FUNCTION_BLOCK PUBLIC ABSTRACT TcoTaskedSequencer EXTENDS TcoCore.TcoSequencerBase
VAR
	{attribute addProperty Name "|[[1]AttributeName]|"}
	{attribute addProperty ToolTip "|[[1]AttributeToolTip]|"}
    _task : TcoInnerTask(THIS^);
    _o    : TcoCore.TcoSequencerObserver(THIS^);	
	
	{attribute addProperty Name "|[[1]Cycle Time Analitics]|"} 
	_cycleTimeAnalitics:CycleTimeAnalitics;	
	_startCleanCycleTime: TIME;
	_stopCleanCycleTime: TIME;
	_timer_1: TON;
	_timer_2: TON;
	_detectStartSeq : R_TRIG;

	_customObserver:TcoCustomSequencerObserver(THIS^);
END_VAR

Run();

PROPERTY PUBLIC AverageCleanCycleTime : TIME
GET
AverageCleanCycleTime:=_cycleTimeAnalitics.AverageCleanCycle;
END_GET
END_PROPERTY

PROPERTY PUBLIC AverageCycleTime : TIME
GET
AverageCycleTime:=_cycleTimeAnalitics.Average;
END_GET
END_PROPERTY

(*~
	<docu>
		<summary>
			Completes the actually running step, when the `inCondition` parameter is `TRUE`.
			Method is typically called inside a step as the transition method.
		</summary>			
	</docu>	
~*)
METHOD PROTECTED FINAL Await
VAR_INPUT
    (*~
	<docu>
		<summary>
			The condition under which the step is completed.
		</summary>			
	</docu>	
~*)
    inCondition : BOOL;
END_VAR
i_StepCompleteWhen(inCondition := inCondition);
END_METHOD

(*~
	<docu>
		<summary>
			<para>
				Completes the sequencer, and return the sequencer pointer to the first step in the seuqence.
				Method is typically called inside the last step of the sequence.
			</para>
		</summary>			
	</docu>	
~*)
METHOD PROTECTED FINAL CompleteSequence



i_CompleteSequence();

IF _cycleTimeAnalitics.FilterConstant = 0 THEN;
	_cycleTimeAnalitics.FilterConstant:=10;
END_IF;


IF _cycleTimeAnalitics.Average = T#0S THEN
	_cycleTimeAnalitics.Average:=_SequenceElapsedTime;
END_IF
_cycleTimeAnalitics.Average:= (((_cycleTimeAnalitics.FilterConstant-1)*_cycleTimeAnalitics.Average)+_LastCycleTime)/_cycleTimeAnalitics.FilterConstant;

_startCleanCycleTime:=T#0S;
_stopCleanCycleTime:=T#0S;
END_METHOD

(*~
	<docu>
		<summary>
			Completes the execution of the current step and moves the sequencer pointer to the next step in order of execution.
			The call returns `ITcoObjectRestorer` that allows to restore object upon step completition.
		</summary>		
		<returns></returns>	
	</docu>	
~*)
METHOD PROTECTED FINAL CompleteStep : ITcoObjectRestorer

CompleteStep := i_CompleteStep();
END_METHOD

PROPERTY CustomObserver : REFERENCE TO TcoCustomSequencerObserver
GET
CustomObserver ref= _customObserver;
END_GET
END_PROPERTY

PROPERTY PUBLIC CycleTimeFilterConstant : UINT
GET
CycleTimeFilterConstant:=_cycleTimeAnalitics.FilterConstant;
END_GET
SET // PUBLIC
_cycleTimeAnalitics.FilterConstant:=CycleTimeFilterConstant;
END_SET
END_PROPERTY

(*~
	<docu>
		<summary>
			Main method of the sequener. Custom code needs to be placed here. The sequencer is executed by call of **Instance.Run()** method.
			This method is abstract, and it must be overridden in derived block.
		</summary>
	</docu>
~*)
METHOD PROTECTED  Main : BOOL
END_METHOD

(*~
	<docu>
		<summary>
			Completes the execution of the current step and moves the sequencer pointer to the next step in order of execution.
			The call returns `ITcoObjectRestorer` that allows to restore object upon step completition.
		</summary>		
		<returns></returns>	
	</docu>	
~*)
METHOD PROTECTED FINAL Next : ITcoObjectRestorer
Next := i_CompleteStep();
END_METHOD

METHOD PUBLIC OnAbort : BOOL
SUPER^.Restore();
END_METHOD

METHOD PUBLIC OnDone : BOOL
END_METHOD

METHOD PUBLIC OnError : BOOL
END_METHOD


(*~
	<docu>
		<summary>
			This method is called on sequence completion (the sequencer's last step was completed). 
			This method can be overridden in derived block with a custom logic.
		</summary>			
	</docu>	
~*)
METHOD PROTECTED OnSequenceCompleted
SUPER^.OnSequenceCompleted();
_customObserver.DefineEndTime(Context.RealTimeClock.NowLocalAsTIMESTRUCT());
_customObserver.CompleteSequence();
END_METHOD

METHOD PUBLIC OnStart
_startCleanCycleTime:=T#0S;
_stopCleanCycleTime:=T#0S;
END_METHOD

(*~
	<docu>
		<summary>
			This method is executed upon step completion.
			This method can be overridden in derived block by custom logic.
		</summary>			
	</docu>	
~*)
METHOD PROTECTED OnStepCompleted


_customObserver.Observe(
	inID:= _currentStep.ID, 
	inDescription:= _currentStep.Description, 
	inDuration:= _currentStep.Duration);
END_METHOD

METHOD pr_Close
VAR_INPUT
END_VAR
_lastClosingCycle := Context.StartCycleCount;

IF _sequencerHasError THEN
    OnSequencerError(_sequencerErrorId);
END_IF

_previousNumberOfStepsInSequence := _numberOfStepsInSequence;
Context.Environment.Messaging.Suspend();

IF _modeController._stepIn.Done THEN
    _modeController._stepIn.Restore();
END_IF

Context.Environment.Messaging.Resume();

_restoringSequence := FALSE;
END_METHOD

METHOD pr_Open
VAR
    _message : STRING(255);
END_VAR
_theOrderOfTheCurrentlyEvaluatedStep := 0;

IF _requestStepActive AND
    _requestedStepId <> (MinStepID - 1) AND
    (_modeController.Mode <> eSequencerMode.StepMode OR _modeController._stepIn.Busy OR _checkStepIdRequestedInStepMode) THEN
    _requestStepCycle := _requestStepCycle + 1;
ELSE
    _requestStepCycle := 0;

END_IF

IF _requestStepCycle > 1 AND NOT _sequencerHasError THEN
    _sequencerErrorId        := eSequencerError.StepWithRequestedIdDoesNotExists;
    _message                 := CONCAT('REQUESTED STEP_ID: ', INT_TO_STRING(_requestedStepId));
    _message                 := CONCAT(_message, ' DOES NOT EXIST');
    _currentStep.Description := _message;
    _currentStep.Status      := eStepStatus.Error;
    THIS^.Messenger.Post(_message, eMessageCategory.ProgrammingError);
    _sequencerHasError := TRUE;

END_IF

IF _StepIdUniquenessControlState = eStepIdUniquenessControlState.NotYetStarted OR
    _StepIdUniquenessControlState = eStepIdUniquenessControlState.Requested THEN
    _StepIdUniquenessControlState := eStepIdUniquenessControlState.Started;

END_IF;

_restoringSequence := FALSE;

_lastOpeningCycle := Context.StartCycleCount;
END_METHOD

(*~
	<docu>
		<summary>
			Terminates the currently executed step and set the sequencer's pointer to the step with Id that corresponds to ```inRequestedStepID``` parameter.
			When the order of the requested step is higher than the order of the currently finished step (the requested step is "after" the current one)
			the requested step is started in the same context cycle.
			When the order of the requested step is lower than the order of the currently finished step (the requested step is "before" the current one)
			the requested step is started in the next context cycle.
			If the requested step is not found even in the next context cycle, the sequencer enters error state ```StepWithRequestedIdDoesNotExists```.
			<para>
				See <see cref="TcoCore.eSequencerError"/> for detailed description.
			</para>
		</summary>
	</docu>
~*)
METHOD PROTECTED FINAL RequestRestoreOrigin : ITcoSequencer

VAR
    _message : STRING(254);
END_VAR
RequestRestoreOrigin := i_RequestStep(inRequestedStepID := RESTORE_STEP_ID);
END_METHOD

(*~
	<docu>
		<summary>
			Terminates the currently executed step and set the sequencer's pointer to the step with Id that corresponds to ```inRequestedStepID``` parameter.
			When the order of the requested step is higher than the order of the currently finished step (the requested step is "after" the current one)
			the requested step is started in the same context cycle.
			When the order of the requested step is lower than the order of the currently finished step (the requested step is "before" the current one)
			the requested step is started in the next context cycle.
			If the requested step is not found even in the next context cycle, the sequencer enters error state ```StepWithRequestedIdDoesNotExists```.
			<para>
				See <see cref="TcoCore.eSequencerError"/> for detailed description.
			</para>
		</summary>
	</docu>
~*)
METHOD PROTECTED FINAL RequestStep : ITcoSequencer
VAR_INPUT
    (*~
		<docu>
			<summary>
				StepId of the step to be executed.
			</summary>
		</docu>
	~*)
    inRequestedStepID : INT := MinStepID - 1;
END_VAR
VAR
    _message : STRING(254);
END_VAR
RequestStep := i_RequestStep(inRequestedStepID := inRequestedStepID);
END_METHOD

(*~
	<docu>
		<summary>
			This method resets the sequencer cycle time . 
				Method is typically called before starting the sequence(e.g.in ground position task) .
		</summary>		
		<returns></returns>	
	</docu>	
~*)
METHOD PUBLIC ResetCycleTime
VAR_INPUT
END_VAR

_cycleTimeAnalitics.Average:=T#0S;
_cycleTimeAnalitics.AverageCleanCycle:=T#0S;
END_METHOD

METHOD PRIVATE ResetTimers
VAR_INPUT
END_VAR
_timer_1.IN:=FALSE;
_timer_2.IN:=FALSE;
END_METHOD

(*~
	<docu>
		<summary>
			<para>
				This method resets the sequencer. 
				Method is typically called before starting the sequence or after error has occured in the sequence.
			</para>
		</summary>			
	</docu>	
~*)
METHOD PUBLIC Restore : ITcoRestorable
SUPER^.Restore();
Task.Restore();
END_METHOD

(*~
	<docu>
		<summary>
			<para>
				Ensures calling the Open(), Main() and Close() methods in the desired order.
				This method is final, so it cannot be overloaded. The **Instance.Run()** needs to be called cyclically inside the appropriate context.
			</para>
		</summary>			
	</docu>	
~*)
METHOD PUBLIC FINAL Run
VAR
    _message : STRING;
END_VAR
IF (_task.Execute()) THEN
    THIS^.pr_Open();

    THIS^.Observer := _o;
    THIS^.Main();
	_detectStartSeq(CLK:=_cycleTimer.ET > T#0S);
    IF _detectStartSeq.Q THEN
        CustomObserver.Clear();
        CustomObserver.DefineStartTime(Context.RealTimeClock.NowLocalAsTIMESTRUCT());
    END_IF

    _customObserver();
    THIS^.pr_Close();
END_IF;
END_METHOD

(*~
	<docu>
		<summary>
			This method s used to start the clean cycle time measurement . 
				Method is typically called at the beggining of the sequence(e.g.in automat sequence) .
		</summary>		
		<returns></returns>	
	</docu>	
~*)

METHOD PUBLIC StartCleanCycleTime
VAR_INPUT
END_VAR
_stopCleanCycleTime:=t#0s;
_startCleanCycleTime:=_SequenceElapsedTime;
END_METHOD

METHOD PROTECTED Step : BOOL
VAR_INPUT
    (*~
	<docu>
		<summary>
			StepId of the current step.
			<remarks>			
				<note type="important">
					This number must be unique throughout the complete sequence.
					It must be a constant or numerical literal and it must not change during the life-time of the sequencer. 
				</note>
			</remarks>
		</summary>		
	</docu>	
~*)
    inStepID : INT;
    (*~
	<docu>
		<summary>
			If this value is false, step body is not executed and execution is moved to the next enabled step.
		</summary>				
	</docu>	
~*)
    inEnabled : BOOL;
    (*~
	<docu>
		<summary>
			Step description text.
		</summary>				
	</docu>	
~*)
    inStepDescription : STRING(254);
END_VAR
Step := i_Step(inStepID := inStepID, inEnabled := inEnabled, inStepDescription := inStepDescription);
END_METHOD

(*~
	<docu>
		<summary>
			Completes the actually running step, when the `inCondition` parameter is `TRUE`.
			Method is typically called inside a step as the transition method.
		</summary>			
	</docu>	
~*)
METHOD PROTECTED FINAL StepCompleteWhen
VAR_INPUT
    (*~
	<docu>
		<summary>
			The condition under which the step is completed.
		</summary>			
	</docu>	
~*)
    inCondition : BOOL;
END_VAR
i_StepCompleteWhen(inCondition := inCondition);
END_METHOD

(*~
	<docu>
		<summary>
			This method s used to stop the clean cycle time measurement . 
				Method is typically called at the end of the sequence(e.g.in automat sequence )  .
		</summary>		
		<returns></returns>	
	</docu>	
~*)

METHOD PUBLIC StopCleanCycleTime
VAR_INPUT
END_VAR

VAR
	cleanCycleTime: TIME;
END_VAR
_stopCleanCycleTime:=_SequenceElapsedTime;

cleanCycleTime:=T#0S;
IF _stopCleanCycleTime>_startCleanCycleTime THEN
	cleanCycleTime:=_stopCleanCycleTime-_startCleanCycleTime;
 END_IF;

IF _cycleTimeAnalitics.FilterConstant = 0 THEN;
	_cycleTimeAnalitics.FilterConstant:=10;
END_IF;


IF _cycleTimeAnalitics.AverageCleanCycle = T#0S THEN
	_cycleTimeAnalitics.AverageCleanCycle:=_stopCleanCycleTime;
END_IF
_cycleTimeAnalitics.AverageCleanCycle:= (((_cycleTimeAnalitics.FilterConstant-1)*_cycleTimeAnalitics.AverageCleanCycle)+cleanCycleTime)/_cycleTimeAnalitics.FilterConstant;
END_METHOD

PROPERTY Task : REFERENCE TO TcoTask
GET
Task REF= _task;
END_GET
END_PROPERTY

METHOD PUBLIC FINAL Timer_1 : BOOL
VAR_INPUT
	Condition : BOOL;
	PT : TIME;
END_VAR
_timer_1(IN:= Condition  and  not IsFreshState, PT:=PT);
Timer_1 := _timer_1.Q;
END_METHOD

METHOD PUBLIC FINAL Timer_2 : BOOL
VAR_INPUT
	Condition : BOOL;
	PT : TIME;
END_VAR
_timer_2(IN:= Condition and not IsFreshState, PT:=PT);
Timer_2 := _timer_2.Q;
END_METHOD

END_FUNCTION_BLOCK

(* stored: Version 1.1.0.1
   POU TcoTaskedSequencer: Id {c1209b3d-cbe5-0fa4-2d35-bd4f0cc6d1e3}, SpecialFunc None
   Folder CycleTimeAnalitics: Id {86c02bf1-155c-0d73-2b05-d09e4bb07f43}
   Folder TaskRelay: Id {afc41ea2-70b7-46a4-8ba7-73e4b0574c74}
   Folder Timers: Id {2af6797e-8e04-46b1-9884-5deb625c01f4}
   Property AverageCleanCycleTime: Id {2856e096-2c70-0832-3dad-a64ad95dfd66}
   Get Get: Id {77b100c9-2a8f-0c53-036a-faa56cf15504}
   Property AverageCycleTime: Id {698abc56-2f06-0ccb-2f4d-dca431ba9514}
   Get Get: Id {99b6ae0d-ed52-0d82-36a8-4c630a7735b6}
   Method Await: Id {12e57bae-9ee5-410f-b614-026e886ed168}
   Method CompleteSequence: Id {e660dda5-e822-0795-15da-43df1875907c}
   Method CompleteStep: Id {16b3254b-2a28-0fb6-2f25-afa0bf333f87}
   Property CustomObserver: Id {763ba8e9-ded2-4f03-904e-ab9953167322}
   Get Get: Id {b06c1ef2-c2bd-4025-9ecc-45fbec14ef9e}
   Property CycleTimeFilterConstant: Id {449ef140-4a3a-0564-3fbc-8b2171d05f79}
   Get Get: Id {731e92ad-ac82-0f37-1645-b8772cd9bfb7}
   Set Set: Id {b34f02a4-fb68-0e7e-294b-d849facfb8bd}
   Method Main: Id {7c01205d-3a68-04f8-3158-3c7d48d004e6}
   Method Next: Id {eafc0316-1e4a-496d-a399-a3f135c3c731}
   Method OnAbort: Id {4a8dbf93-63ad-425f-a385-076450b1741f}
   Method OnDone: Id {30fb0e8a-1cb0-4f9e-a2ec-ea455b994447}
   Method OnError: Id {0ad4a5a1-079e-4d8c-ab31-9475260ad3db}
   Method OnSequenceCompleted: Id {e4d81d54-4428-4634-8a18-7e1c98a10d56}
   Method OnStart: Id {3f6df8fb-4ab1-4f1c-90a2-1116dcabff12}
   Method OnStepCompleted: Id {59491651-e455-40c4-8ccf-cceff7ff9eb5}
   Method pr_Close: Id {f8eb2d85-b3ce-4599-b36f-51273583184e}
   Method pr_Open: Id {8c53ec29-7192-431b-a895-8408067229d4}
   Method RequestRestoreOrigin: Id {1f323207-31e2-4052-b838-44e4d33d526b}
   Method RequestStep: Id {05e23ca1-6a4e-00c5-0fd4-d50792c02a3f}
   Method ResetCycleTime: Id {fcf27ed1-9cd7-0c2b-3a39-1e54bf3bc4ac}
   Method ResetTimers: Id {c0e378a0-09f3-4f5d-8221-03bde2a0ef7b}
   Method Restore: Id {a3c44169-c865-41a7-b04d-fb6593fd4c0f}
   Method Run: Id {18d5420d-14f4-0ac5-255d-8d8a78d1e1c6}
   Method StartCleanCycleTime: Id {1d853ffc-17de-0de5-037b-8f202c4d5f30}
   Method Step: Id {c3c5f2f3-742a-0ae5-3d6d-5a15b5bc9906}
   Method StepCompleteWhen: Id {bd441a6f-affd-05d6-027c-c88ec0339cbb}
   Method StopCleanCycleTime: Id {c24139e5-8cd2-0fb9-0cad-ad76beab6e9f}
   Property Task: Id {31b22691-83dc-0d45-2152-2f03cc6b6a6e}
   Get Get: Id {6c191508-6ada-00b4-2005-7e4c80b0377a}
   Method Timer_1: Id {1124a7d8-f03e-48d1-8410-80f26add3bdf}
   Method Timer_2: Id {ba7678b2-3bdc-4bb3-9f5e-196bf9a8fe98} *)
